LIN {X 0,Y 27.582,Z 393.876,A -85,B 0,C 180,E1 -30315.238,E2 -30315.238} C_VEL
LIN {X 0,Y 27.102,Z 394.041,A -85,B 0,C 180,E1 -30330,E2 -30330} C_VEL
LIN {X 0,Y 27.584,Z 393.876,A -85,B 0,C 180,E1 -30344.761,E2 -30344.761} C_VEL
LIN {X 0,Y 29.577,Z 393.274,A -85,B 0,C 180,E1 -30358.374,E2 -30358.374} C_VEL
LIN {X 0,Y 37.282,Z 390.804,A -85,B 0,C 180,E1 -30378.94,E2 -30378.94} C_VEL
LIN {X 0,Y 45.184,Z 387.846,A -85,B 0,C 180,E1 -30388.81,E2 -30388.81} C_VEL
LIN {X 0,Y 53.994,Z 383.852,A -85,B 0,C 180,E1 -30395.661,E2 -30395.661} C_VEL
LIN {X 0,Y 63.452,Z 378.635,A -85,B 0,C 180,E1 -30400.704,E2 -30400.704} C_VEL
LIN {X 0,Y 68.089,Z 375.76,A -85,B 0,C 180,E1 -30402.698,E2 -30402.698} C_VEL
LIN {X 0,Y 69.59,Z 374.593,A -85,B 0,C 180,E1 -30403.619,E2 -30403.619} C_VEL
LIN {X 0,Y 71.545,Z 372.845,A -85,B 0,C 180,E1 -30405.754,E2 -30405.754} C_VEL
LIN {X 0,Y 72.575,Z 371.53,A -85,B 0,C 180,E1 -30408.801,E2 -30408.801} C_VEL
LIN {X 0,Y 73.697,Z 369.853,A -85,B 0,C 180,E1 -30414.496,E2 -30414.496} C_VEL
LIN {X 0,Y 74.428,Z 368.818,A -85,B 0,C 180,E1 -30419.969,E2 -30419.969} C_VEL
LIN {X 0,Y 73.406,Z 369.697,A -85,B 0,C 180,E1 -30426.657,E2 -30426.657} C_VEL
LIN {X 0,Y 72.495,Z 371.18,A -85,B 0,C 180,E1 -30434.204,E2 -30434.204} C_VEL
LIN {X 0,Y 72.187,Z 371.886,A -85,B 0,C 180,E1 -30436.947,E2 -30436.947} C_VEL
LIN {X 0,Y 71.541,Z 372.997,A -85,B 0,C 180,E1 -30440.074,E2 -30440.074} C_VEL
LIN {X 0,Y 70.136,Z 375.286,A -85,B 0,C 180,E1 -30445.601,E2 -30445.601} C_VEL
LIN {X 0,Y 68.3,Z 377.668,A -85,B 0,C 180,E1 -30450.922,E2 -30450.922} C_VEL
LIN {X 0,Y 65.911,Z 380.469,A -85,B 0,C 180,E1 -30456.898,E2 -30456.898} C_VEL
LIN {X 0,Y 62.64,Z 384.563,A -85,B 0,C 180,E1 -30467.688,E2 -30467.688} C_VEL
LIN {X 0,Y 61.841,Z 386.777,A -85,B 0,C 180,E1 -30475.374,E2 -30475.374} C_VEL
LIN {X 0,Y 62.411,Z 388.638,A -85,B 0,C 180,E1 -30484.178,E2 -30484.178} C_VEL
LIN {X 0,Y 67.05,Z 390.548,A -85,B 0,C 180,E1 -30497.899,E2 -30497.899} C_VEL
LIN {X 0,Y 71.26,Z 390.972,A -85,B 0,C 180,E1 -30504.34,E2 -30504.34} C_VEL
LIN {X 0,Y 76.437,Z 390.96,A -85,B 0,C 180,E1 -30510,E2 -30510} C_VEL
LIN {X 0,Y 70.68,Z 390.918,A -85,B 0,C 180,E1 -30516.436,E2 -30516.436} C_VEL
LIN {X 0,Y 65.549,Z 390.19,A -85,B 0,C 180,E1 -30525.362,E2 -30525.362} C_VEL
LIN {X 0,Y 62.305,Z 388.42,A -85,B 0,C 180,E1 -30536.82,E2 -30536.82} C_VEL
LIN {X 0,Y 61.952,Z 386.011,A -85,B 0,C 180,E1 -30547.497,E2 -30547.497} C_VEL
LIN {X 0,Y 64.482,Z 382.101,A -85,B 0,C 180,E1 -30559.211,E2 -30559.211} C_VEL
LIN {X 0,Y 67.324,Z 378.895,A -85,B 0,C 180,E1 -30566.628,E2 -30566.628} C_VEL
LIN {X 0,Y 69.62,Z 375.97,A -85,B 0,C 180,E1 -30572.769,E2 -30572.769} C_VEL
LIN {X 0,Y 70.725,Z 374.381,A -85,B 0,C 180,E1 -30576.617,E2 -30576.617} C_VEL
LIN {X 0,Y 71.535,Z 373.001,A -85,B 0,C 180,E1 -30579.924,E2 -30579.924} C_VEL
LIN {X 0,Y 72.16,Z 371.904,A -85,B 0,C 180,E1 -30583.046,E2 -30583.046} C_VEL
LIN {X 0,Y 72.862,Z 370.492,A -85,B 0,C 180,E1 -30588.911,E2 -30588.911} C_VEL
LIN {X 0,Y 73.623,Z 369.484,A -85,B 0,C 180,E1 -30594.555,E2 -30594.555} C_VEL
LIN {X 0,Y 74.426,Z 368.82,A -85,B 0,C 180,E1 -30600.031,E2 -30600.031} C_VEL
LIN {X 0,Y 73.474,Z 370.092,A -85,B 0,C 180,E1 -30606.183,E2 -30606.183} C_VEL
LIN {X 0,Y 72.29,Z 371.209,A -85,B 0,C 180,E1 -30608.322,E2 -30608.322} C_VEL
LIN {X 0,Y 69.842,Z 373.127,A -85,B 0,C 180,E1 -30610.251,E2 -30610.251} C_VEL
LIN {X 0,Y 67.349,Z 374.892,A -85,B 0,C 180,E1 -30611.399,E2 -30611.399} C_VEL
LIN {X 0,Y 57.525,Z 380.665,A -85,B 0,C 180,E1 -30614.433,E2 -30614.433} C_VEL
LIN {X 0,Y 48.231,Z 385.171,A -85,B 0,C 180,E1 -30618.714,E2 -30618.714} C_VEL
LIN {X 0,Y 38.883,Z 388.787,A -85,B 0,C 180,E1 -30625.348,E2 -30625.348} C_VEL
LIN {X 0,Y 33.037,Z 390.592,A -85,B 0,C 180,E1 -30631.688,E2 -30631.688} C_VEL
LIN {X 0,Y 23.55,Z 393.062,A -85,B 0,C 180,E1 -30653.356,E2 -30653.356} C_VEL
LIN {X 0,Y 20.788,Z 393.665,A -85,B 0,C 180,E1 -30670.24,E2 -30670.24} C_VEL
LIN {X 0,Y 20.009,Z 393.83,A -85,B 0,C 180,E1 -30690,E2 -30690} C_VEL
LIN {X 0,Y 20.789,Z 393.665,A -85,B 0,C 180,E1 -30709.758,E2 -30709.758} C_VEL
LIN {X 0,Y 23.552,Z 393.062,A -85,B 0,C 180,E1 -30726.641,E2 -30726.641} C_VEL
LIN {X 0,Y 33.036,Z 390.592,A -85,B 0,C 180,E1 -30748.313,E2 -30748.313} C_VEL
LIN {X 0,Y 41.938,Z 387.634,A -85,B 0,C 180,E1 -30757.174,E2 -30757.174} C_VEL
LIN {X 0,Y 51.471,Z 383.641,A -85,B 0,C 180,E1 -30762.9,E2 -30762.9} C_VEL
LIN {X 0,Y 61.316,Z 378.506,A -85,B 0,C 180,E1 -30766.953,E2 -30766.953} C_VEL
LIN {X 0,Y 64.64,Z 376.585,A -85,B 0,C 180,E1 -30768.1,E2 -30768.1} C_VEL
LIN {X 0,Y 66.819,Z 374.789,A -85,B 0,C 180,E1 -30771.22,E2 -30771.22} C_VEL
LIN {X 0,Y 67.397,Z 374.048,A -85,B 0,C 180,E1 -30773.98,E2 -30773.98} C_VEL
LIN {X 0,Y 68.442,Z 372.913,A -85,B 0,C 180,E1 -30779.966,E2 -30779.966} C_VEL
LIN {X 0,Y 67.496,Z 373.56,A -85,B 0,C 180,E1 -30785.942,E2 -30785.942} C_VEL
LIN {X 0,Y 66.668,Z 374.63,A -85,B 0,C 180,E1 -30792.135,E2 -30792.135} C_VEL
LIN {X 0,Y 65.965,Z 375.631,A -85,B 0,C 180,E1 -30796.492,E2 -30796.492} C_VEL
LIN {X 0,Y 64.306,Z 377.526,A -85,B 0,C 180,E1 -30802.449,E2 -30802.449} C_VEL
LIN {X 0,Y 62.859,Z 379.16,A -85,B 0,C 180,E1 -30806.564,E2 -30806.564} C_VEL
LIN {X 0,Y 61.235,Z 380.719,A -85,B 0,C 180,E1 -30810.598,E2 -30810.598} C_VEL
LIN {X 0,Y 58.668,Z 383.105,A -85,B 0,C 180,E1 -30816.743,E2 -30816.743} C_VEL
LIN {X 0,Y 55.196,Z 387.024,A -85,B 0,C 180,E1 -30830.459,E2 -30830.459} C_VEL
LIN {X 0,Y 55.183,Z 389.317,A -85,B 0,C 180,E1 -30842.962,E2 -30842.962} C_VEL
LIN {X 0,Y 58.532,Z 390.808,A -85,B 0,C 180,E1 -30856.105,E2 -30856.105} C_VEL
LIN {X 0,Y 63.443,Z 391.319,A -85,B 0,C 180,E1 -30865.06,E2 -30865.06} C_VEL
LIN {X 0,Y 67.421,Z 391.228,A -85,B 0,C 180,E1 -30870,E2 -30870} C_VEL
LIN {X 0,Y 62.471,Z 391.235,A -85,B 0,C 180,E1 -30876.459,E2 -30876.459} C_VEL
LIN {X 0,Y 58.168,Z 390.736,A -85,B 0,C 180,E1 -30885.025,E2 -30885.025} C_VEL
LIN {X 0,Y 54.905,Z 388.671,A -85,B 0,C 180,E1 -30900.797,E2 -30900.797} C_VEL
LIN {X 0,Y 55.844,Z 385.951,A -85,B 0,C 180,E1 -30913.796,E2 -30913.796} C_VEL
LIN {X 0,Y 59.619,Z 382.188,A -85,B 0,C 180,E1 -30925.604,E2 -30925.604} C_VEL
LIN {X 0,Y 61.227,Z 380.719,A -85,B 0,C 180,E1 -30929.415,E2 -30929.415} C_VEL
LIN {X 0,Y 62.881,Z 379.137,A -85,B 0,C 180,E1 -30933.488,E2 -30933.488} C_VEL
LIN {X 0,Y 64.319,Z 377.518,A -85,B 0,C 180,E1 -30937.556,E2 -30937.556} C_VEL
LIN {X 0,Y 65.963,Z 375.631,A -85,B 0,C 180,E1 -30943.512,E2 -30943.512} C_VEL
LIN {X 0,Y 66.662,Z 374.634,A -85,B 0,C 180,E1 -30947.864,E2 -30947.864} C_VEL
LIN {X 0,Y 67.488,Z 373.565,A -85,B 0,C 180,E1 -30954.058,E2 -30954.058} C_VEL
LIN {X 0,Y 68.428,Z 372.922,A -85,B 0,C 180,E1 -30960.034,E2 -30960.034} C_VEL
LIN {X 0,Y 67.352,Z 374.078,A -85,B 0,C 180,E1 -30966.024,E2 -30966.024} C_VEL
LIN {X 0,Y 66.804,Z 374.801,A -85,B 0,C 180,E1 -30968.792,E2 -30968.792} C_VEL
LIN {X 0,Y 64.645,Z 376.585,A -85,B 0,C 180,E1 -30971.921,E2 -30971.921} C_VEL
LIN {X 0,Y 57.525,Z 380.665,A -85,B 0,C 180,E1 -30974.433,E2 -30974.433} C_VEL
LIN {X 0,Y 52.314,Z 383.14,A -85,B 0,C 180,E1 -30975.88,E2 -30975.88} C_VEL
LIN {X 0,Y 46.805,Z 385.407,A -85,B 0,C 180,E1 -30976.522,E2 -30976.522} C_VEL
LIN {X 0,Y 35.461,Z 388.953,A -85,B 0,C 180,E1 -30977.62,E2 -30977.62} C_VEL
LIN {X 0,Y 29.019,Z 390.638,A -85,B 0,C 180,E1 -30980.92,E2 -30980.92} C_VEL
LIN {X 0,Y 28.156,Z 390.771,A -85,B 0,C 180,E1 -30981.79,E2 -30981.79} C_VEL
LIN {X 0,Y 18.339,Z 392.85,A -85,B 0,C 180,E1 -30999.965,E2 -30999.965} C_VEL
LIN {X 0,Y 14.289,Z 393.453,A -85,B 0,C 180,E1 -31020.539,E2 -31020.539} C_VEL
LIN {X 0,Y 12.906,Z 393.619,A -85,B 0,C 180,E1 -31050,E2 -31050} C_VEL
LIN {X 0,Y 14.29,Z 393.453,A -85,B 0,C 180,E1 -31079.458,E2 -31079.458} C_VEL
LIN {X 0,Y 18.34,Z 392.85,A -85,B 0,C 180,E1 -31100.032,E2 -31100.032} C_VEL
LIN {X 0,Y 29.912,Z 390.379,A -85,B 0,C 180,E1 -31120.019,E2 -31120.019} C_VEL
LIN {X 0,Y 39.719,Z 387.422,A -85,B 0,C 180,E1 -31126.695,E2 -31126.695} C_VEL
LIN {X 0,Y 49.84,Z 383.428,A -85,B 0,C 180,E1 -31130.771,E2 -31130.771} C_VEL
LIN {X 0,Y 60.106,Z 378.293,A -85,B 0,C 180,E1 -31133.617,E2 -31133.617} C_VEL
LIN {X 0,Y 61.568,Z 377.261,A -85,B 0,C 180,E1 -31136.69,E2 -31136.69} C_VEL
LIN {X 0,Y 62.204,Z 376.756,A -85,B 0,C 180,E1 -31139.962,E2 -31139.962} C_VEL
LIN {X 0,Y 61.139,Z 377.341,A -85,B 0,C 180,E1 -31146.562,E2 -31146.562} C_VEL
LIN {X 0,Y 60.007,Z 378.428,A -85,B 0,C 180,E1 -31153.506,E2 -31153.506} C_VEL
LIN {X 0,Y 58.98,Z 379.466,A -85,B 0,C 180,E1 -31157.588,E2 -31157.588} C_VEL
LIN {X 0,Y 57.636,Z 380.604,A -85,B 0,C 180,E1 -31161.413,E2 -31161.413} C_VEL
LIN {X 0,Y 55.286,Z 382.439,A -85,B 0,C 180,E1 -31167.148,E2 -31167.148} C_VEL
LIN {X 0,Y 51.715,Z 385.051,A -85,B 0,C 180,E1 -31175.376,E2 -31175.376} C_VEL
LIN {X 0,Y 48.773,Z 387.571,A -85,B 0,C 180,E1 -31186.022,E2 -31186.022} C_VEL
LIN {X 0,Y 48.215,Z 390.16,A -85,B 0,C 180,E1 -31204.069,E2 -31204.069} C_VEL
LIN {X 0,Y 50.764,Z 391.149,A -85,B 0,C 180,E1 -31215.521,E2 -31215.521} C_VEL
LIN {X 0,Y 56.262,Z 391.563,A -85,B 0,C 180,E1 -31226.891,E2 -31226.891} C_VEL
LIN {X 0,Y 58.459,Z 391.495,A -85,B 0,C 180,E1 -31230,E2 -31230} C_VEL
LIN {X 0,Y 53.747,Z 391.496,A -85,B 0,C 180,E1 -31237.513,E2 -31237.513} C_VEL
LIN {X 0,Y 50.282,Z 391.062,A -85,B 0,C 180,E1 -31246.233,E2 -31246.233} C_VEL
LIN {X 0,Y 48.012,Z 389.87,A -85,B 0,C 180,E1 -31258.673,E2 -31258.673} C_VEL
LIN {X 0,Y 49.112,Z 387.27,A -85,B 0,C 180,E1 -31275.683,E2 -31275.683} C_VEL
LIN {X 0,Y 53.18,Z 384.069,A -85,B 0,C 180,E1 -31288.142,E2 -31288.142} C_VEL
LIN {X 0,Y 55.272,Z 382.44,A -85,B 0,C 180,E1 -31292.879,E2 -31292.879} C_VEL
LIN {X 0,Y 57.646,Z 380.599,A -85,B 0,C 180,E1 -31298.591,E2 -31298.591} C_VEL
LIN {X 0,Y 58.981,Z 379.466,A -85,B 0,C 180,E1 -31302.408,E2 -31302.408} C_VEL
LIN {X 0,Y 60.004,Z 378.43,A -85,B 0,C 180,E1 -31306.494,E2 -31306.494} C_VEL
LIN {X 0,Y 61.134,Z 377.344,A -85,B 0,C 180,E1 -31313.438,E2 -31313.438} C_VEL
LIN {X 0,Y 62.195,Z 376.762,A -85,B 0,C 180,E1 -31320.038,E2 -31320.038} C_VEL
LIN {X 0,Y 61.547,Z 377.273,A -85,B 0,C 180,E1 -31323.311,E2 -31323.311} C_VEL
LIN {X 0,Y 60.106,Z 378.293,A -85,B 0,C 180,E1 -31326.385,E2 -31326.385} C_VEL
LIN {X 0,Y 49.841,Z 383.428,A -85,B 0,C 180,E1 -31329.233,E2 -31329.233} C_VEL
LIN {X 0,Y 39.72,Z 387.422,A -85,B 0,C 180,E1 -31333.308,E2 -31333.308} C_VEL
LIN {X 0,Y 29.912,Z 390.379,A -85,B 0,C 180,E1 -31339.982,E2 -31339.982} C_VEL
LIN {X 0,Y 28.156,Z 390.771,A -85,B 0,C 180,E1 -31341.79,E2 -31341.79} C_VEL
LIN {X 0,Y 22.873,Z 391.906,A -85,B 0,C 180,E1 -31347.289,E2 -31347.289} C_VEL
LIN {X 0,Y 17.383,Z 392.746,A -85,B 0,C 180,E1 -31353.417,E2 -31353.417} C_VEL
LIN {X 0,Y 7.304,Z 393.434,A -85,B 0,C 180,E1 -31386.727,E2 -31386.727} C_VEL
LIN {X 0,Y 7.414,Z 393.289,A -85,B 0,C 180,E1 -31452.514,E2 -31452.514} C_VEL
LIN {X 0,Y 14.812,Z 392.638,A -85,B 0,C 180,E1 -31481.615,E2 -31481.615} C_VEL
LIN {X 0,Y 28.281,Z 390.167,A -85,B 0,C 180,E1 -31493.716,E2 -31493.716} C_VEL
LIN {X 0,Y 38.706,Z 387.21,A -85,B 0,C 180,E1 -31497.016,E2 -31497.016} C_VEL
LIN {X 0,Y 49.202,Z 383.216,A -85,B 0,C 180,E1 -31499.005,E2 -31499.005} C_VEL
LIN {X 0,Y 55.764,Z 380.243,A -85,B 0,C 180,E1 -31499.958,E2 -31499.958} C_VEL
LIN {X 0,Y 54.477,Z 380.86,A -85,B 0,C 180,E1 -31507.368,E2 -31507.368} C_VEL
LIN {X 0,Y 52.639,Z 382.095,A -85,B 0,C 180,E1 -31515.44,E2 -31515.44} C_VEL
LIN {X 0,Y 51.703,Z 382.717,A -85,B 0,C 180,E1 -31517.918,E2 -31517.918} C_VEL
LIN {X 0,Y 49.628,Z 384.095,A -85,B 0,C 180,E1 -31522.649,E2 -31522.649} C_VEL
LIN {X 0,Y 43.78,Z 387.514,A -85,B 0,C 180,E1 -31536.618,E2 -31536.618} C_VEL
LIN {X 0,Y 41.479,Z 389.167,A -85,B 0,C 180,E1 -31547.333,E2 -31547.333} C_VEL
LIN {X 0,Y 42.084,Z 391.319,A -85,B 0,C 180,E1 -31570.489,E2 -31570.489} C_VEL
LIN {X 0,Y 45.055,Z 391.758,A -85,B 0,C 180,E1 -31581.026,E2 -31581.026} C_VEL
LIN {X 0,Y 49.606,Z 391.758,A -85,B 0,C 180,E1 -31590,E2 -31590} C_VEL
LIN {X 0,Y 43.418,Z 391.539,A -85,B 0,C 180,E1 -31604.023,E2 -31604.023} C_VEL
LIN {X 0,Y 40.847,Z 390.409,A -85,B 0,C 180,E1 -31621.075,E2 -31621.075} C_VEL
LIN {X 0,Y 42.512,Z 388.272,A -85,B 0,C 180,E1 -31638.679,E2 -31638.679} C_VEL
LIN {X 0,Y 48.005,Z 384.978,A -85,B 0,C 180,E1 -31654.003,E2 -31654.003} C_VEL
LIN {X 0,Y 49.622,Z 384.096,A -85,B 0,C 180,E1 -31657.359,E2 -31657.359} C_VEL
LIN {X 0,Y 51.705,Z 382.716,A -85,B 0,C 180,E1 -31662.074,E2 -31662.074} C_VEL
LIN {X 0,Y 52.644,Z 382.093,A -85,B 0,C 180,E1 -31664.561,E2 -31664.561} C_VEL
LIN {X 0,Y 54.473,Z 380.861,A -85,B 0,C 180,E1 -31672.631,E2 -31672.631} C_VEL
LIN {X 0,Y 55.759,Z 380.246,A -85,B 0,C 180,E1 -31680.042,E2 -31680.042} C_VEL
LIN {X 0,Y 45.698,Z 384.748,A -85,B 0,C 180,E1 -31681.556,E2 -31681.556} C_VEL
LIN {X 0,Y 35.221,Z 388.363,A -85,B 0,C 180,E1 -31683.902,E2 -31683.902} C_VEL
LIN {X 0,Y 25.562,Z 390.72,A -85,B 0,C 180,E1 -31687.671,E2 -31687.671} C_VEL
LIN {X 0,Y 14.811,Z 392.638,A -85,B 0,C 180,E1 -31698.381,E2 -31698.381} C_VEL
LIN {X 0,Y 8.821,Z 393.241,A -85,B 0,C 180,E1 -31717.183,E2 -31717.183} C_VEL
LIN {X 0,Y 5.794,Z 393.407,A -85,B 0,C 180,E1 -31770,E2 -31770} C_VEL
LIN {X 0,Y 7.414,Z 393.289,A -85,B 0,C 180,E1 -31812.514,E2 -31812.514} C_VEL
LIN {X 0,Y 10.131,Z 393.107,A -85,B 0,C 180,E1 -31831.324,E2 -31831.324} C_VEL
LIN {X 0,Y 16.434,Z 392.316,A -85,B 0,C 180,E1 -31852.284,E2 -31852.284} C_VEL
LIN {X 0,Y 27.107,Z 390.283,A -85,B 0,C 180,E1 -31865.766,E2 -31865.766} C_VEL
LIN {X 0,Y 32.797,Z 388.84,A -85,B 0,C 180,E1 -31867.664,E2 -31867.664} C_VEL
LIN {X 0,Y 34.717,Z 388.339,A -85,B 0,C 180,E1 -31867.697,E2 -31867.697} C_VEL
LIN {X 0,Y 42.53,Z 385.777,A -85,B 0,C 180,E1 -31867.494,E2 -31867.494} C_VEL
LIN {X 0,Y 47.293,Z 384.046,A -85,B 0,C 180,E1 -31868.495,E2 -31868.495} C_VEL
LIN {X 0,Y 44.157,Z 385.552,A -85,B 0,C 180,E1 -31877.265,E2 -31877.265} C_VEL
LIN {X 0,Y 39.448,Z 387.758,A -85,B 0,C 180,E1 -31887.03,E2 -31887.03} C_VEL
LIN {X 0,Y 35.819,Z 389.414,A -85,B 0,C 180,E1 -31898.296,E2 -31898.296} C_VEL
LIN {X 0,Y 34.225,Z 391.57,A -85,B 0,C 180,E1 -31925.752,E2 -31925.752} C_VEL
LIN {X 0,Y 36.602,Z 392.013,A -85,B 0,C 180,E1 -31938.93,E2 -31938.93} C_VEL
LIN {X 0,Y 40.855,Z 392.019,A -85,B 0,C 180,E1 -31950,E2 -31950} C_VEL
LIN {X 0,Y 36.062,Z 391.933,A -85,B 0,C 180,E1 -31963.284,E2 -31963.284} C_VEL
LIN {X 0,Y 33.805,Z 390.99,A -85,B 0,C 180,E1 -31983.866,E2 -31983.866} C_VEL
LIN {X 0,Y 36.628,Z 388.975,A -85,B 0,C 180,E1 -32004.937,E2 -32004.937} C_VEL
LIN {X 0,Y 39.45,Z 387.758,A -85,B 0,C 180,E1 -32012.967,E2 -32012.967} C_VEL
LIN {X 0,Y 44.156,Z 385.552,A -85,B 0,C 180,E1 -32022.738,E2 -32022.738} C_VEL
LIN {X 0,Y 47.293,Z 384.046,A -85,B 0,C 180,E1 -32031.504,E2 -32031.504} C_VEL
LIN {X 0,Y 42.53,Z 385.777,A -85,B 0,C 180,E1 -32032.51,E2 -32032.51} C_VEL
LIN {X 0,Y 35.455,Z 388.151,A -85,B 0,C 180,E1 -32032.347,E2 -32032.347} C_VEL
LIN {X 0,Y 28.398,Z 389.955,A -85,B 0,C 180,E1 -32031.855,E2 -32031.855} C_VEL
LIN {X 0,Y 14.271,Z 392.426,A -85,B 0,C 180,E1 -32030.029,E2 -32030.029} C_VEL
LIN {X 0,Y 7.254,Z 393.029,A -85,B 0,C 180,E1 -32025.653,E2 -32025.653} C_VEL
LIN {X 0,Y 1.304,Z 393.196,A -85,B 0,C 180,E1 -31950,E2 -31950} C_VEL
LIN {X 0,Y 7.254,Z 393.029,A -85,B 0,C 180,E1 -31874.338,E2 -31874.338} C_VEL
LIN {X 0,Y 14.271,Z 392.426,A -85,B 0,C 180,E1 -31869.967,E2 -31869.967} C_VEL
LIN {X 0,Y 28.398,Z 389.955,A -85,B 0,C 180,E1 -31868.147,E2 -31868.147} C_VEL
LIN {X 0,Y 34.717,Z 388.339,A -85,B 0,C 180,E1 -31867.697,E2 -31867.697} C_VEL
LIN {X 0,Y 35.33,Z 388.191,A -85,B 0,C 180,E1 -31868.759,E2 -31868.759} C_VEL
LIN {X 0,Y 35.276,Z 388.247,A -85,B 0,C 180,E1 -31871.968,E2 -31871.968} C_VEL
LIN {X 0,Y 34.036,Z 388.673,A -85,B 0,C 180,E1 -31877.268,E2 -31877.268} C_VEL
LIN {X 0,Y 29.856,Z 390.22,A -85,B 0,C 180,E1 -31890.862,E2 -31890.862} C_VEL
LIN {X 0,Y 27.399,Z 391.165,A -85,B 0,C 180,E1 -31905.136,E2 -31905.136} C_VEL
LIN {X 0,Y 28.269,Z 392.267,A -85,B 0,C 180,E1 -31935.605,E2 -31935.605} C_VEL
LIN {X 0,Y 32.213,Z 392.276,A -85,B 0,C 180,E1 -31950,E2 -31950} C_VEL
LIN {X 0,Y 28.319,Z 392.266,A -85,B 0,C 180,E1 -31964.369,E2 -31964.369} C_VEL
LIN {X 0,Y 26.906,Z 391.545,A -85,B 0,C 180,E1 -31988.551,E2 -31988.551} C_VEL
LIN {X 0,Y 32.959,Z 389.103,A -85,B 0,C 180,E1 -32017.59,E2 -32017.59} C_VEL
LIN {X 0,Y 30.238,Z 389.744,A -85,B 0,C 180,E1 -32018.386,E2 -32018.386} C_VEL
LIN {X 0,Y 17.027,Z 392.213,A -85,B 0,C 180,E1 -32005.641,E2 -32005.641} C_VEL
LIN {X 0,Y 11.355,Z 392.817,A -85,B 0,C 180,E1 -31988.236,E2 -31988.236} C_VEL
LIN {X 0,Y 8.393,Z 392.985,A -85,B 0,C 180,E1 -31950,E2 -31950} C_VEL
LIN {X 0,Y 11.355,Z 392.817,A -85,B 0,C 180,E1 -31911.761,E2 -31911.761} C_VEL
LIN {X 0,Y 17.026,Z 392.213,A -85,B 0,C 180,E1 -31894.357,E2 -31894.357} C_VEL
LIN {X 0,Y 30.238,Z 389.744,A -85,B 0,C 180,E1 -31881.615,E2 -31881.615} C_VEL
LIN {X 0,Y 32.96,Z 389.104,A -85,B 0,C 180,E1 -31882.431,E2 -31882.431} C_VEL
LIN {X 0,Y 27.399,Z 391.165,A -85,B 0,C 180,E1 -31905.136,E2 -31905.136} C_VEL
LIN {X 0,Y 26.047,Z 391.587,A -85,B 0,C 180,E1 -31909.934,E2 -31909.934} C_VEL
LIN {X 0,Y 20.519,Z 392.353,A -85,B 0,C 180,E1 -31922.73,E2 -31922.73} C_VEL
LIN {X 0,Y 20.131,Z 392.507,A -85,B 0,C 180,E1 -31928.971,E2 -31928.971} C_VEL
LIN {X 0,Y 23.585,Z 392.533,A -85,B 0,C 180,E1 -31950,E2 -31950} C_VEL
LIN {X 0,Y 19.777,Z 392.378,A -85,B 0,C 180,E1 -31977.859,E2 -31977.859} C_VEL
LIN {X 0,Y 17.505,Z 392.605,A -85,B 0,C 180,E1 -31973.671,E2 -31973.671} C_VEL
LIN {X 0,Y 15.502,Z 392.773,A -85,B 0,C 180,E1 -31950,E2 -31950} C_VEL
LIN {X 0,Y 17.504,Z 392.605,A -85,B 0,C 180,E1 -31926.328,E2 -31926.328} C_VEL
LIN {X 0,Y 19.768,Z 392.379,A -85,B 0,C 180,E1 -31922.128,E2 -31922.128} C_VEL
LIN {X 0,Y 20.131,Z 392.507,A -85,B 0,C 180,E1 -31928.971,E2 -31928.971} C_VEL
LIN {X 0,Y 20.61,Z 394.504,A -85,B 0,C 180,E1 -31934.126,E2 -31934.126} C_VEL
LIN {X 0,Y 20.61,Z 600,A -85,B 0,C 180,E1 -31934.126,E2 -31934.126} C_VEL
LIN {X 0,Y 20.61,Z 600,A -85,B 0,C 180,E1 -31934.126,E2 -31934.126}

QRS_NEXT_CUT()

QRS_NEXT()
QRS_HOME()

END
